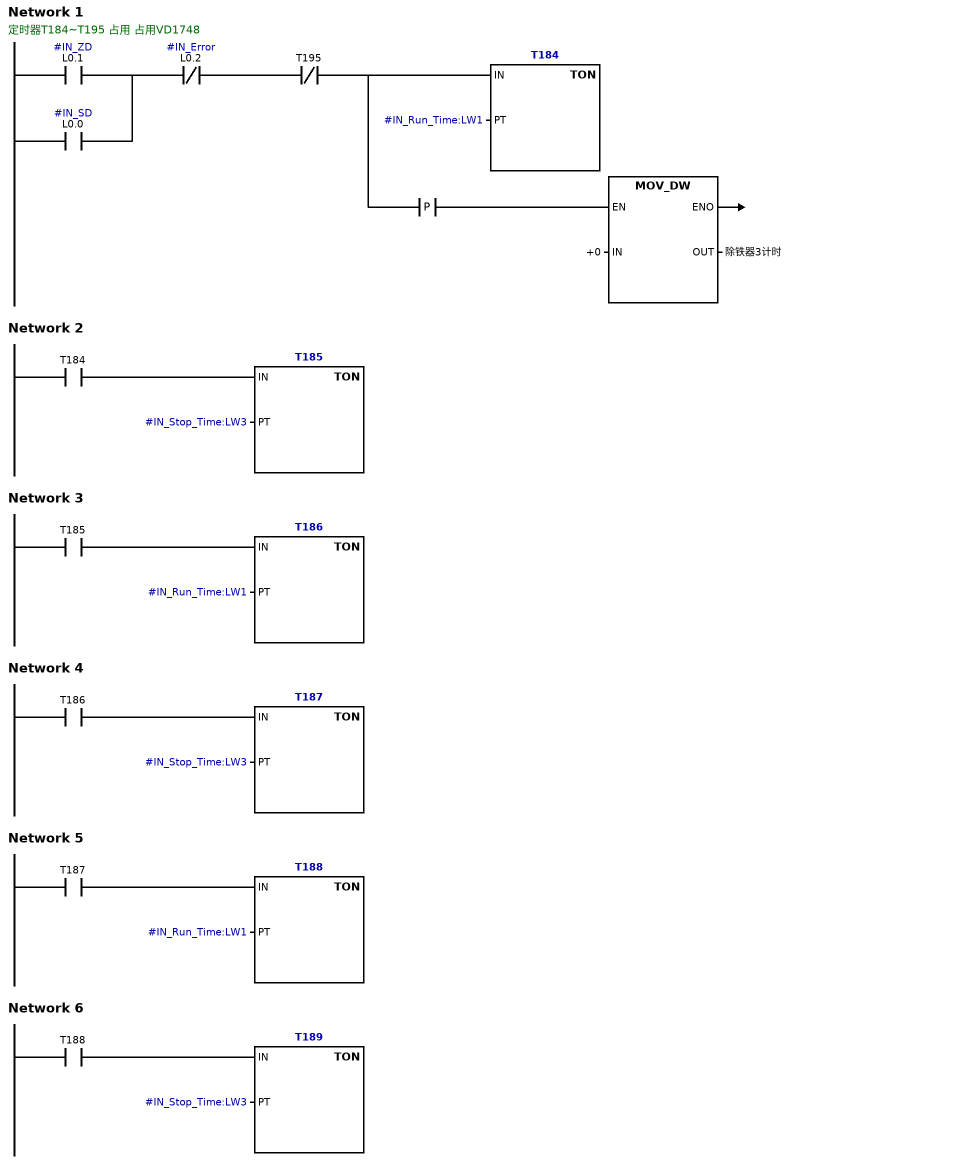
[picture p168: SBR79 networks 1-6]
Network 1
// 定时器T184~T195 占用 占用VD1748
// (network saved uncompiled; LAD cells follow)
// row 0: c0 -| |- #IN_ZD:L0.1 v  c1 -|/|- #IN_Error:L0.2  c2 -|/|- T195 v  c3 --  c4 [TON T184 IN:=power@row0, PT:=#IN_Run_Time:LW1]
// row 1: c0 -| |- #IN_SD:L0.0 ^  c2 ^v  c4 [box]
// row 2: c2 ^  c3 -|P|-  c4 --  c5 [MOV_DW EN:=power@row2, IN:=+0, ENO=>power, OUT=>除铁器3计时]  c6 ->
// row 3: c5 [box]
Network 2
LD     T184
TON    T185, #IN_Stop_Time:LW3
Network 3
LD     T185
TON    T186, #IN_Run_Time:LW1
Network 4
LD     T186
TON    T187, #IN_Stop_Time:LW3
Network 5
LD     T187
TON    T188, #IN_Run_Time:LW1
Network 6
LD     T188
TON    T189, #IN_Stop_Time:LW3
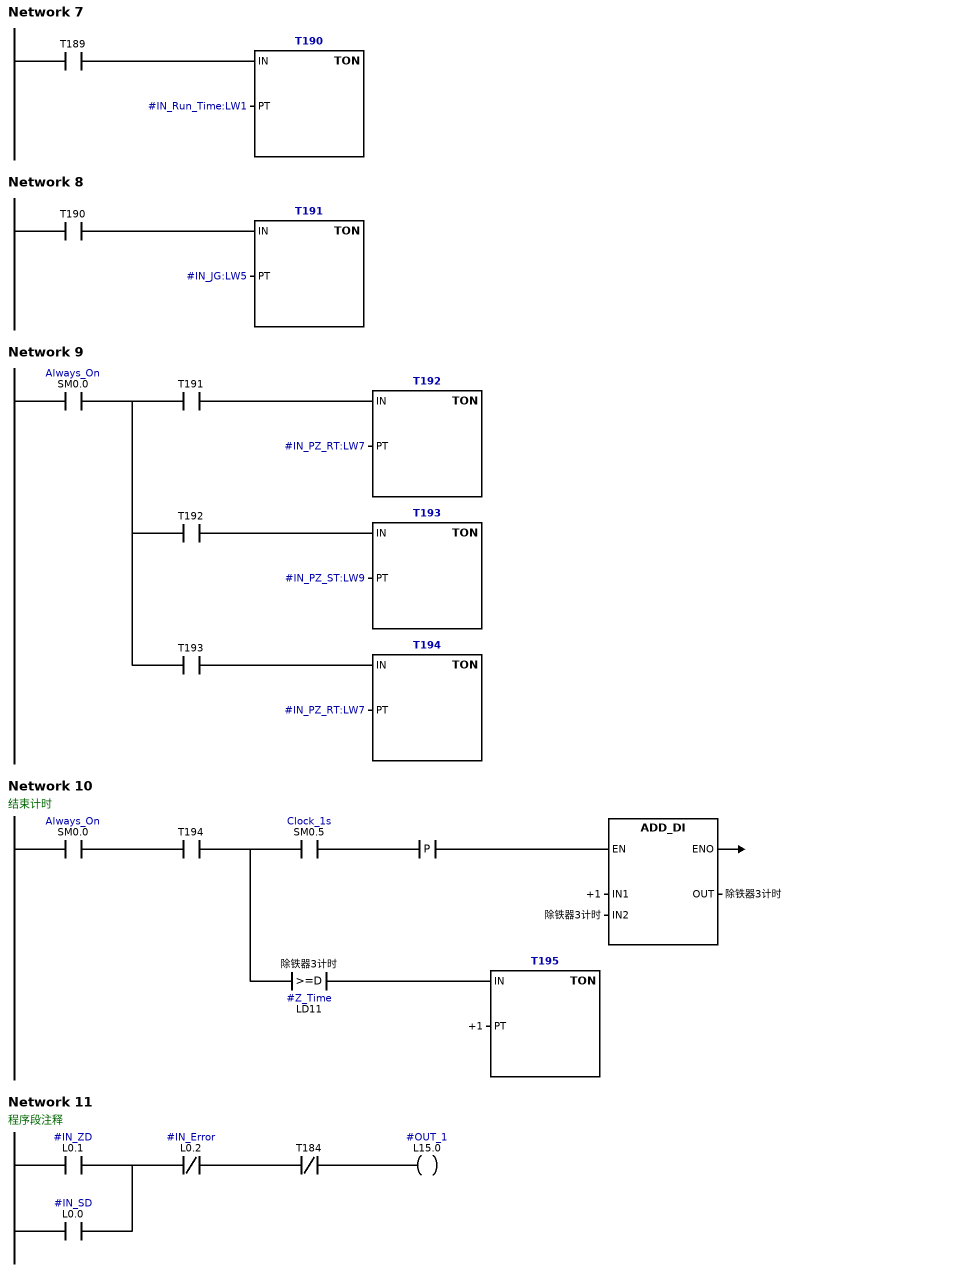
Network 7
LD     T189
TON    T190, #IN_Run_Time:LW1
Network 8
LD     T190
TON    T191, #IN_JG:LW5
Network 9
LD     Always_On:SM0.0
LPS
A      T191
TON    T192, #IN_PZ_RT:LW7
LRD
A      T192
TON    T193, #IN_PZ_ST:LW9
LPP
A      T193
TON    T194, #IN_PZ_RT:LW7
Network 10
// 结束计时
// (network saved uncompiled; LAD cells follow)
// row 0: c0 -| |- Always_On:SM0.0  c1 -| |- T194 v  c2 -| |- Clock_1s:SM0.5  c3 -|P|-  c4 --  c5 [ADD_DI EN:=power@row0, IN1:=+1, IN2:=除铁器3计时, ENO=>power, OUT=>除铁器3计时]  c6 ->
// row 1: c1 ^v  c5 [box]
// row 2: c1 ^  c2 -|>=D|- 除铁器3计时, #Z_Time:LD11  c3 --  c4 [TON T195 IN:=power@row2, PT:=+1]
// row 3: c4 [box]
Network 11
//  程序段注释
LD     #IN_ZD:L0.1
O      #IN_SD:L0.0
AN     #IN_Error:L0.2
AN     T184
=      #OUT_1:L15.0
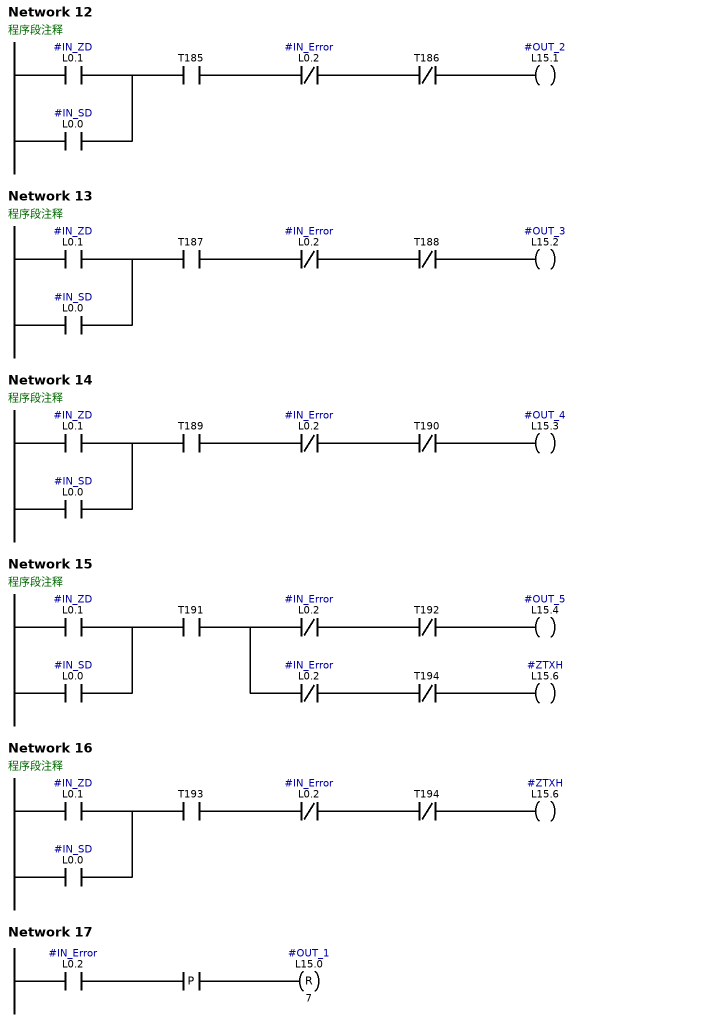
Network 12
//  程序段注释
LD     #IN_ZD:L0.1
O      #IN_SD:L0.0
A      T185
AN     #IN_Error:L0.2
AN     T186
=      #OUT_2:L15.1
Network 13
//  程序段注释
LD     #IN_ZD:L0.1
O      #IN_SD:L0.0
A      T187
AN     #IN_Error:L0.2
AN     T188
=      #OUT_3:L15.2
Network 14
//  程序段注释
LD     #IN_ZD:L0.1
O      #IN_SD:L0.0
A      T189
AN     #IN_Error:L0.2
AN     T190
=      #OUT_4:L15.3
Network 15
//  程序段注释
LD     #IN_ZD:L0.1
O      #IN_SD:L0.0
A      T191
LPS
AN     #IN_Error:L0.2
AN     T192
=      #OUT_5:L15.4
LPP
AN     #IN_Error:L0.2
AN     T194
=      #ZTXH:L15.6
Network 16
//  程序段注释
LD     #IN_ZD:L0.1
O      #IN_SD:L0.0
A      T193
AN     #IN_Error:L0.2
AN     T194
=      #ZTXH:L15.6
Network 17
LD     #IN_Error:L0.2
EU
R      #OUT_1:L15.0, 7
END_SUBROUTINE_BLOCK

SUBROUTINE_BLOCK 脉冲阀4组1:SBR80
TITLE=
VAR_INPUT
IN_SD:BOOL;	// L0.0 
IN_ZD:BOOL;	// L0.1 
IN_Error:BOOL;	// L0.2 
IN_Run_Time:INT;	// LW1 
IN_Stop_Time:INT;	// LW3 
END_VAR
VAR_OUTPUT
OUT_1:BOOL;	// L5.0 
OUT_2:BOOL;	// L5.1 
OUT_3:BOOL;	// L5.2 
OUT_4:BOOL;	// L5.3 
END_VAR
VAR
TP1:BOOL;	// L5.4 
TP2:BOOL;	// L5.5 
END_VAR
BEGIN
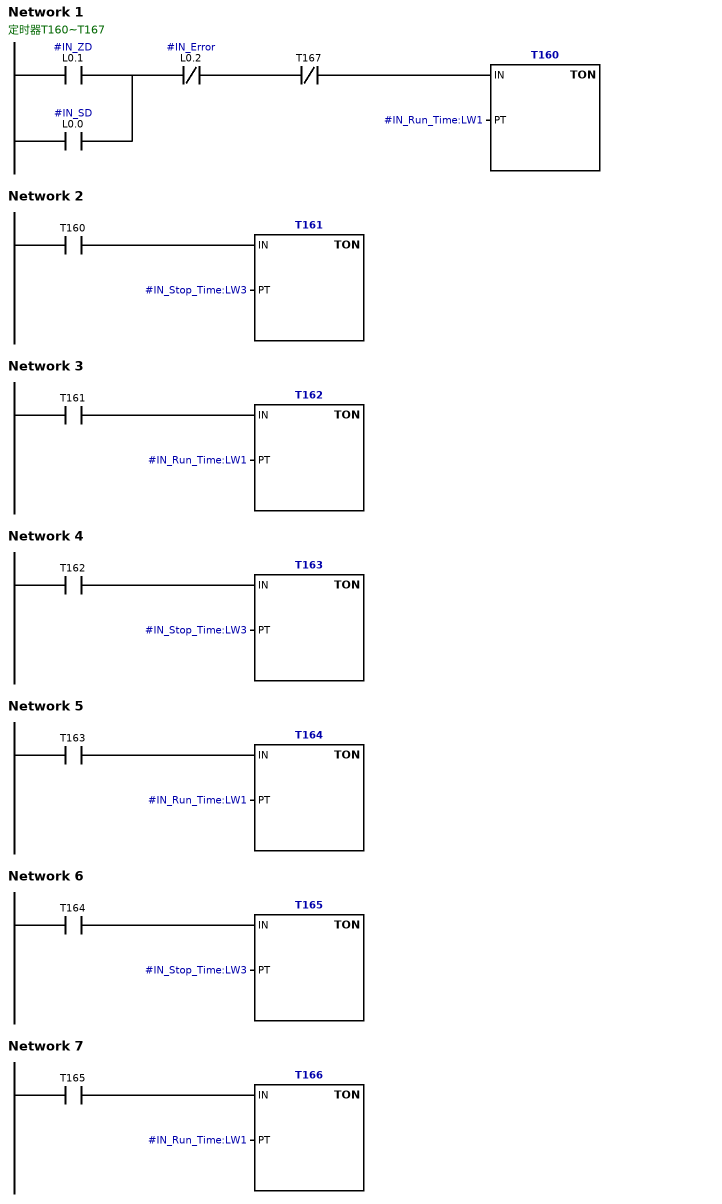
Network 1
// 定时器T160~T167
LD     #IN_ZD:L0.1
O      #IN_SD:L0.0
AN     #IN_Error:L0.2
AN     T167
TON    T160, #IN_Run_Time:LW1
Network 2
LD     T160
TON    T161, #IN_Stop_Time:LW3
Network 3
LD     T161
TON    T162, #IN_Run_Time:LW1
Network 4
LD     T162
TON    T163, #IN_Stop_Time:LW3
Network 5
LD     T163
TON    T164, #IN_Run_Time:LW1
Network 6
LD     T164
TON    T165, #IN_Stop_Time:LW3
Network 7
LD     T165
TON    T166, #IN_Run_Time:LW1
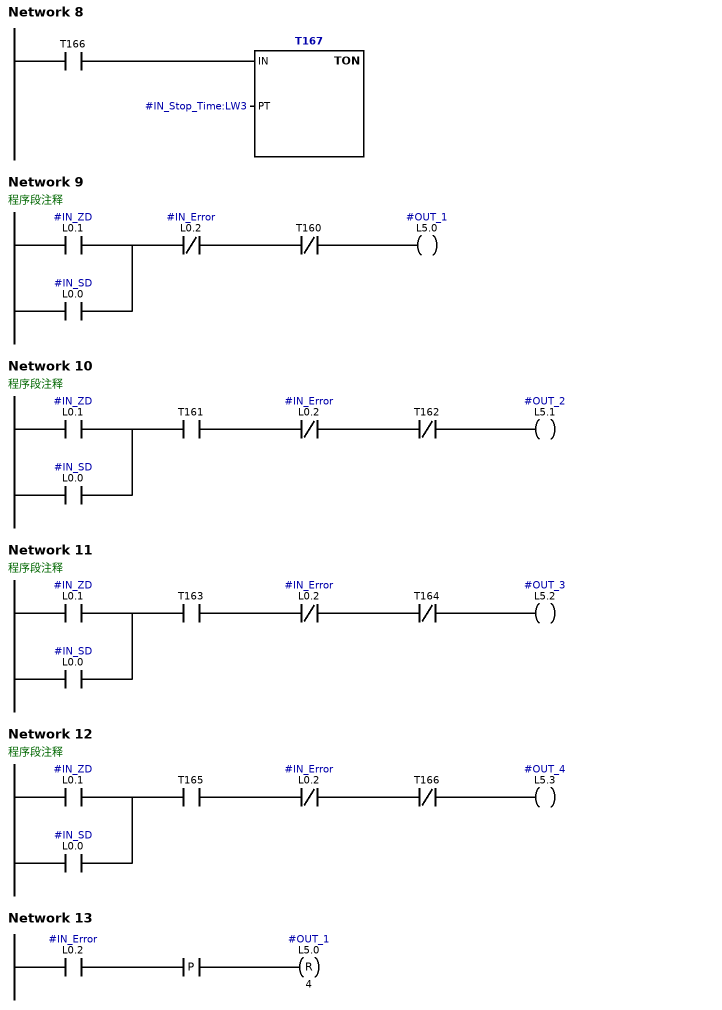
Network 8
LD     T166
TON    T167, #IN_Stop_Time:LW3
Network 9
//  程序段注释
LD     #IN_ZD:L0.1
O      #IN_SD:L0.0
AN     #IN_Error:L0.2
AN     T160
=      #OUT_1:L5.0
Network 10
//  程序段注释
LD     #IN_ZD:L0.1
O      #IN_SD:L0.0
A      T161
AN     #IN_Error:L0.2
AN     T162
=      #OUT_2:L5.1
Network 11
//  程序段注释
LD     #IN_ZD:L0.1
O      #IN_SD:L0.0
A      T163
AN     #IN_Error:L0.2
AN     T164
=      #OUT_3:L5.2
Network 12
//  程序段注释
LD     #IN_ZD:L0.1
O      #IN_SD:L0.0
A      T165
AN     #IN_Error:L0.2
AN     T166
=      #OUT_4:L5.3
Network 13
LD     #IN_Error:L0.2
EU
R      #OUT_1:L5.0, 4
END_SUBROUTINE_BLOCK

SUBROUTINE_BLOCK 脉冲阀4组2:SBR81
TITLE=
VAR_INPUT
IN_SD:BOOL;	// L0.0 
IN_ZD:BOOL;	// L0.1 
IN_Error:BOOL;	// L0.2 
IN_Run_Time:INT;	// LW1 
IN_Stop_Time:INT;	// LW3 
END_VAR
VAR_OUTPUT
OUT_1:BOOL;	// L5.0 
OUT_2:BOOL;	// L5.1 
OUT_3:BOOL;	// L5.2 
OUT_4:BOOL;	// L5.3 
END_VAR
VAR
TP1:BOOL;	// L5.4 
TP2:BOOL;	// L5.5 
END_VAR
BEGIN
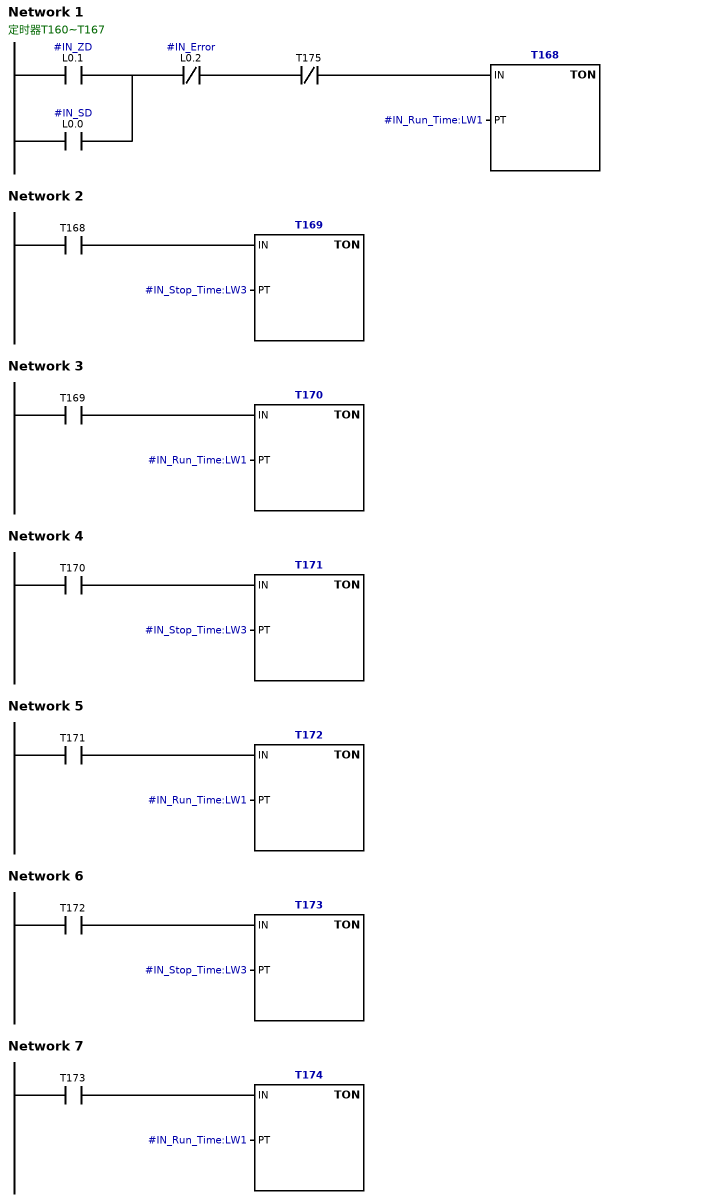
Network 1
// 定时器T160~T167
LD     #IN_ZD:L0.1
O      #IN_SD:L0.0
AN     #IN_Error:L0.2
AN     T175
TON    T168, #IN_Run_Time:LW1
Network 2
LD     T168
TON    T169, #IN_Stop_Time:LW3
Network 3
LD     T169
TON    T170, #IN_Run_Time:LW1
Network 4
LD     T170
TON    T171, #IN_Stop_Time:LW3
Network 5
LD     T171
TON    T172, #IN_Run_Time:LW1
Network 6
LD     T172
TON    T173, #IN_Stop_Time:LW3
Network 7
LD     T173
TON    T174, #IN_Run_Time:LW1
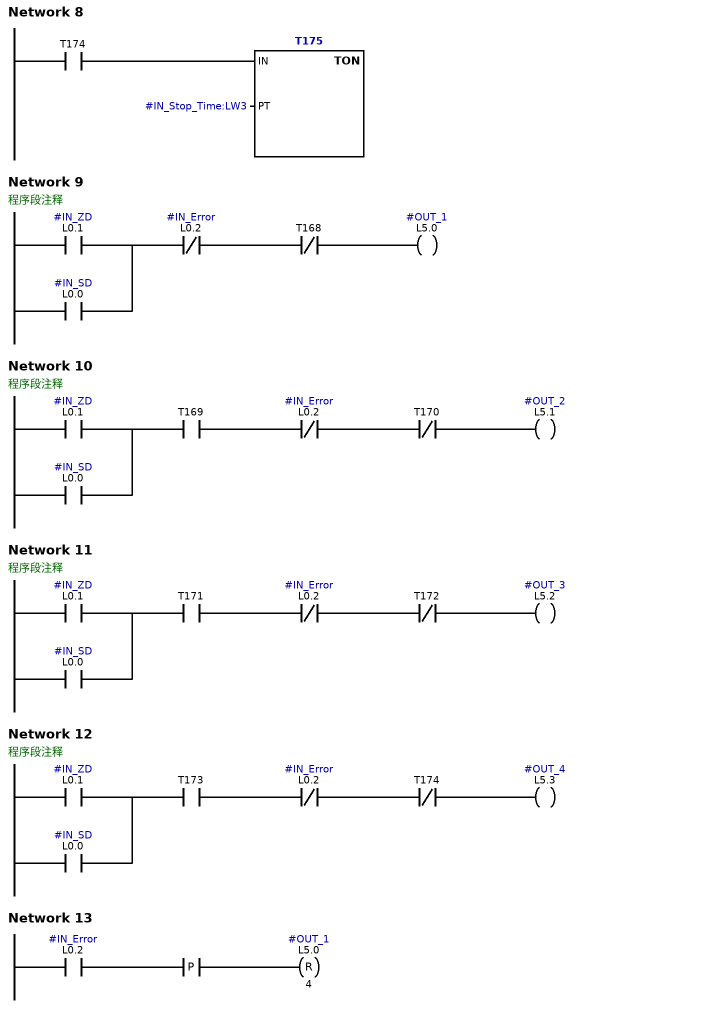
Network 8
LD     T174
TON    T175, #IN_Stop_Time:LW3
Network 9
//  程序段注释
LD     #IN_ZD:L0.1
O      #IN_SD:L0.0
AN     #IN_Error:L0.2
AN     T168
=      #OUT_1:L5.0
Network 10
//  程序段注释
LD     #IN_ZD:L0.1
O      #IN_SD:L0.0
A      T169
AN     #IN_Error:L0.2
AN     T170
=      #OUT_2:L5.1
Network 11
//  程序段注释
LD     #IN_ZD:L0.1
O      #IN_SD:L0.0
A      T171
AN     #IN_Error:L0.2
AN     T172
=      #OUT_3:L5.2
Network 12
//  程序段注释
LD     #IN_ZD:L0.1
O      #IN_SD:L0.0
A      T173
AN     #IN_Error:L0.2
AN     T174
=      #OUT_4:L5.3
Network 13
LD     #IN_Error:L0.2
EU
R      #OUT_1:L5.0, 4
END_SUBROUTINE_BLOCK

SUBROUTINE_BLOCK 脉冲阀4组3:SBR82
TITLE=
VAR_INPUT
IN_SD:BOOL;	// L0.0 
IN_ZD:BOOL;	// L0.1 
IN_Error:BOOL;	// L0.2 
IN_Run_Time:INT;	// LW1 
IN_Stop_Time:INT;	// LW3 
END_VAR
VAR_OUTPUT
OUT_1:BOOL;	// L5.0 
OUT_2:BOOL;	// L5.1 
OUT_3:BOOL;	// L5.2 
OUT_4:BOOL;	// L5.3 
END_VAR
VAR
TP1:BOOL;	// L5.4 
TP2:BOOL;	// L5.5 
END_VAR
BEGIN
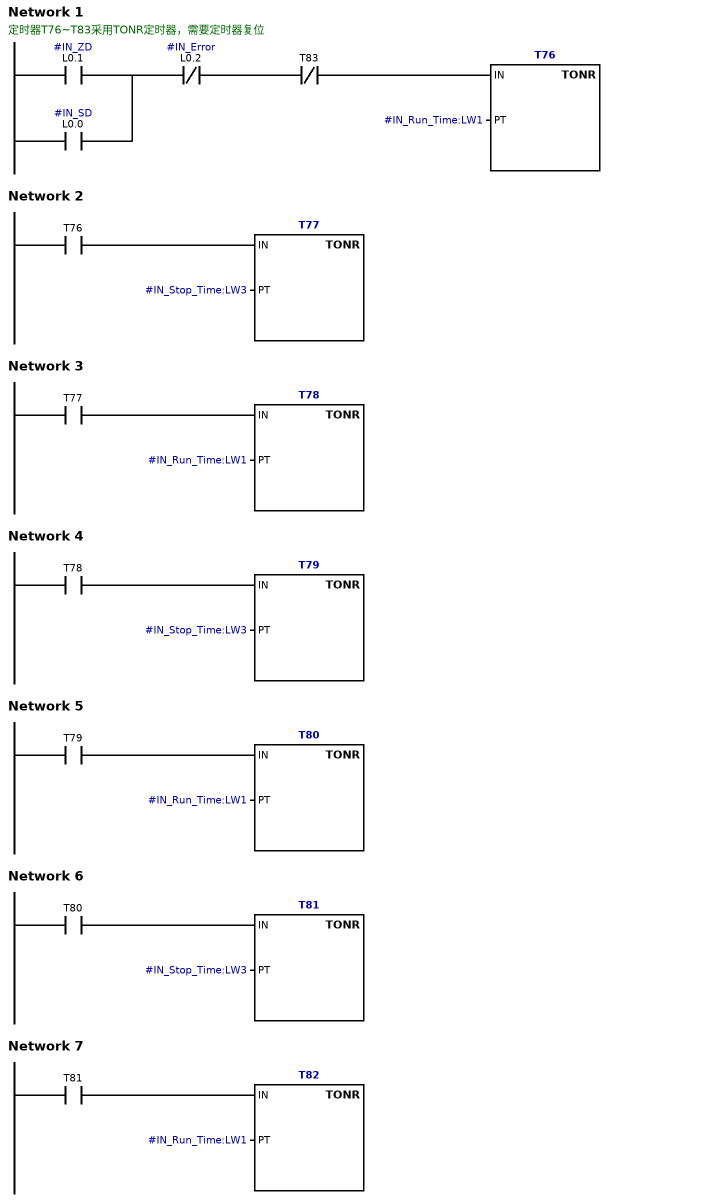
Network 1
// 定时器T76~T83采用TONR定时器，需要定时器复位
LD     #IN_ZD:L0.1
O      #IN_SD:L0.0
AN     #IN_Error:L0.2
AN     T83
TONR   T76, #IN_Run_Time:LW1
Network 2
LD     T76
TONR   T77, #IN_Stop_Time:LW3
Network 3
LD     T77
TONR   T78, #IN_Run_Time:LW1
Network 4
LD     T78
TONR   T79, #IN_Stop_Time:LW3
Network 5
LD     T79
TONR   T80, #IN_Run_Time:LW1
Network 6
LD     T80
TONR   T81, #IN_Stop_Time:LW3
Network 7
LD     T81
TONR   T82, #IN_Run_Time:LW1
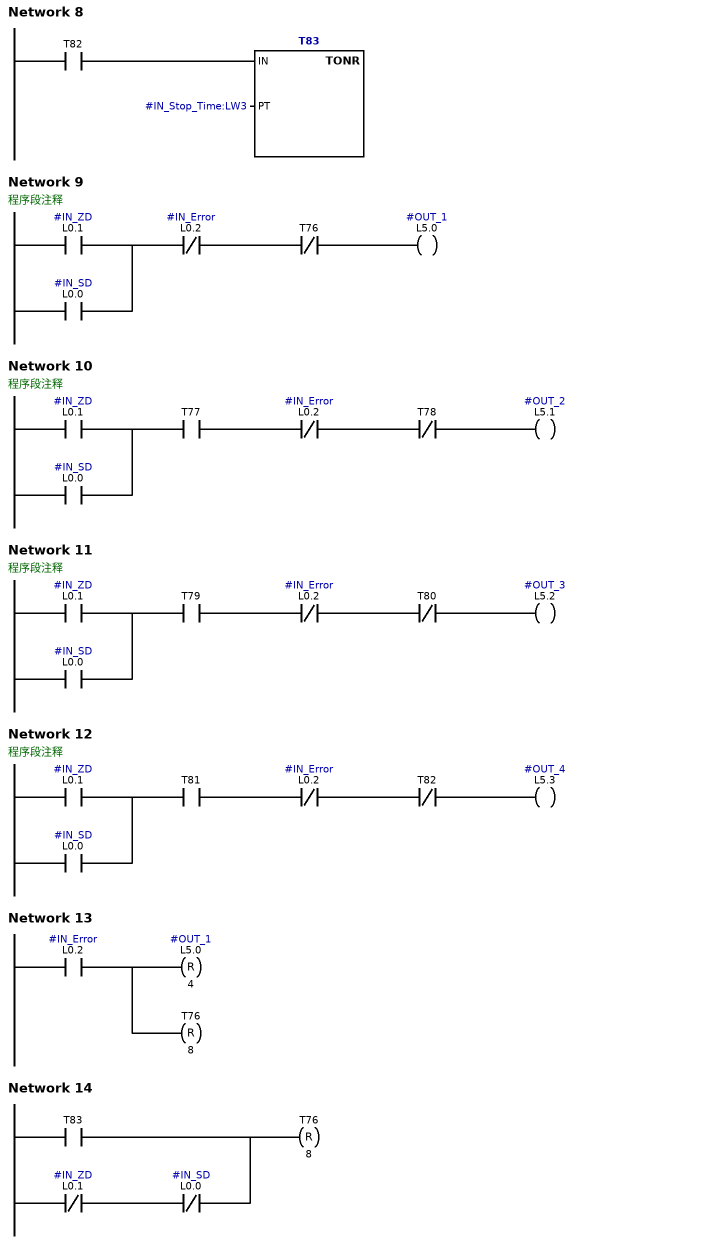
Network 8
LD     T82
TONR   T83, #IN_Stop_Time:LW3
Network 9
//  程序段注释
LD     #IN_ZD:L0.1
O      #IN_SD:L0.0
AN     #IN_Error:L0.2
AN     T76
=      #OUT_1:L5.0
Network 10
//  程序段注释
LD     #IN_ZD:L0.1
O      #IN_SD:L0.0
A      T77
AN     #IN_Error:L0.2
AN     T78
=      #OUT_2:L5.1
Network 11
//  程序段注释
LD     #IN_ZD:L0.1
O      #IN_SD:L0.0
A      T79
AN     #IN_Error:L0.2
AN     T80
=      #OUT_3:L5.2
Network 12
//  程序段注释
LD     #IN_ZD:L0.1
O      #IN_SD:L0.0
A      T81
AN     #IN_Error:L0.2
AN     T82
=      #OUT_4:L5.3
Network 13
LD     #IN_Error:L0.2
R      #OUT_1:L5.0, 4
R      T76, 8
Network 14
LD     T83
LDN    #IN_ZD:L0.1
AN     #IN_SD:L0.0
OLD
R      T76, 8
END_SUBROUTINE_BLOCK

SUBROUTINE_BLOCK 脉冲阀4组4:SBR83
TITLE=
VAR_INPUT
IN_SD:BOOL;	// L0.0 
IN_ZD:BOOL;	// L0.1 
IN_Error:BOOL;	// L0.2 
IN_Run_Time:INT;	// LW1 
IN_Stop_Time:INT;	// LW3 
END_VAR
VAR_OUTPUT
OUT_1:BOOL;	// L5.0 
OUT_2:BOOL;	// L5.1 
OUT_3:BOOL;	// L5.2 
OUT_4:BOOL;	// L5.3 
END_VAR
VAR
TP1:BOOL;	// L5.4 
TP2:BOOL;	// L5.5 
END_VAR
BEGIN
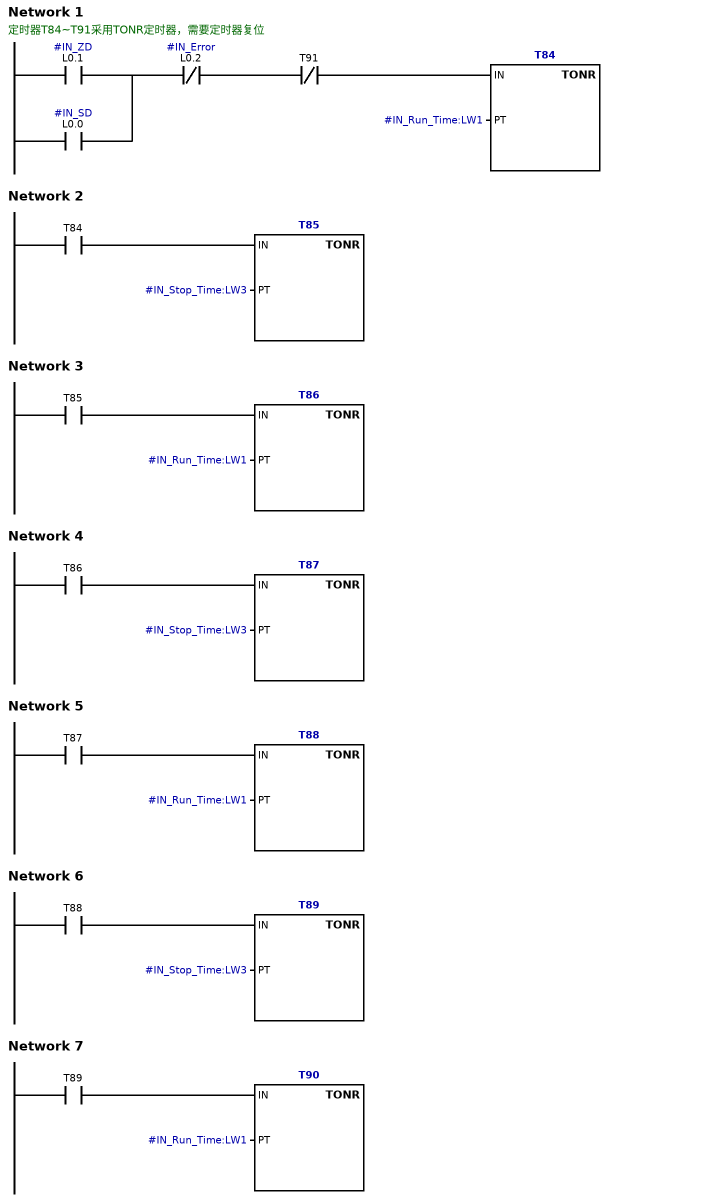
Network 1
// 定时器T84~T91采用TONR定时器，需要定时器复位
LD     #IN_ZD:L0.1
O      #IN_SD:L0.0
AN     #IN_Error:L0.2
AN     T91
TONR   T84, #IN_Run_Time:LW1
Network 2
LD     T84
TONR   T85, #IN_Stop_Time:LW3
Network 3
LD     T85
TONR   T86, #IN_Run_Time:LW1
Network 4
LD     T86
TONR   T87, #IN_Stop_Time:LW3
Network 5
LD     T87
TONR   T88, #IN_Run_Time:LW1
Network 6
LD     T88
TONR   T89, #IN_Stop_Time:LW3
Network 7
LD     T89
TONR   T90, #IN_Run_Time:LW1
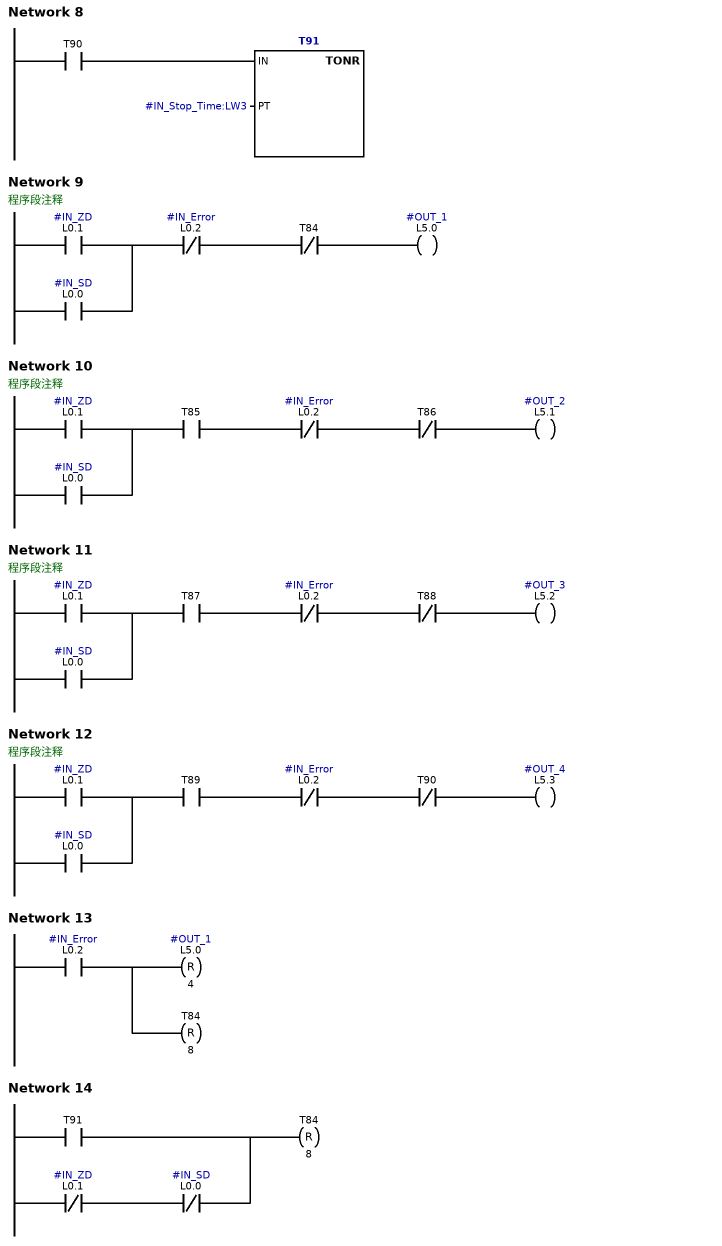
Network 8
LD     T90
TONR   T91, #IN_Stop_Time:LW3
Network 9
//  程序段注释
LD     #IN_ZD:L0.1
O      #IN_SD:L0.0
AN     #IN_Error:L0.2
AN     T84
=      #OUT_1:L5.0
Network 10
//  程序段注释
LD     #IN_ZD:L0.1
O      #IN_SD:L0.0
A      T85
AN     #IN_Error:L0.2
AN     T86
=      #OUT_2:L5.1
Network 11
//  程序段注释
LD     #IN_ZD:L0.1
O      #IN_SD:L0.0
A      T87
AN     #IN_Error:L0.2
AN     T88
=      #OUT_3:L5.2
Network 12
//  程序段注释
LD     #IN_ZD:L0.1
O      #IN_SD:L0.0
A      T89
AN     #IN_Error:L0.2
AN     T90
=      #OUT_4:L5.3
Network 13
LD     #IN_Error:L0.2
R      #OUT_1:L5.0, 4
R      T84, 8
Network 14
LD     T91
LDN    #IN_ZD:L0.1
AN     #IN_SD:L0.0
OLD
R      T84, 8
END_SUBROUTINE_BLOCK

SUBROUTINE_BLOCK 脉冲阀4组5:SBR84
TITLE=
VAR_INPUT
IN_SD:BOOL;	// L0.0 
IN_ZD:BOOL;	// L0.1 
IN_Error:BOOL;	// L0.2 
IN_Run_Time:INT;	// LW1 
IN_Stop_Time:INT;	// LW3 
END_VAR
VAR_OUTPUT
OUT_1:BOOL;	// L5.0 
OUT_2:BOOL;	// L5.1 
OUT_3:BOOL;	// L5.2 
OUT_4:BOOL;	// L5.3 
END_VAR
VAR
TP1:BOOL;	// L5.4 
TP2:BOOL;	// L5.5 
END_VAR
BEGIN
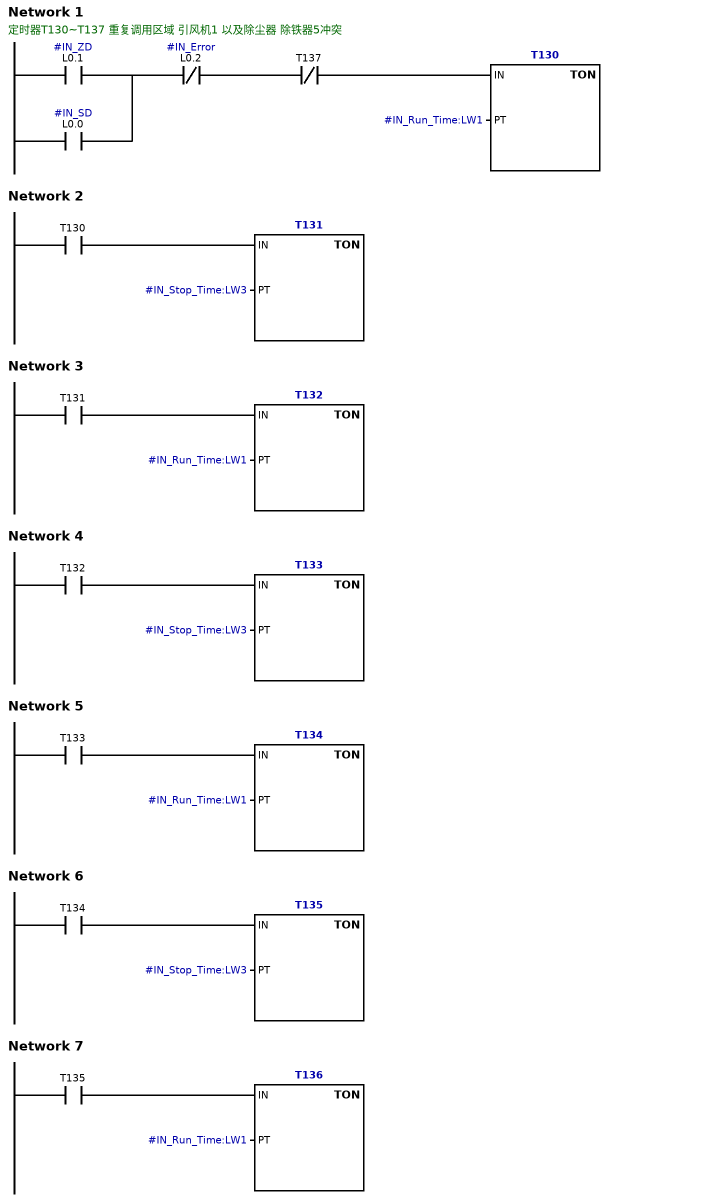
Network 1
// 定时器T130~T137 重复调用区域 引风机1 以及除尘器 除铁器5冲突
LD     #IN_ZD:L0.1
O      #IN_SD:L0.0
AN     #IN_Error:L0.2
AN     T137
TON    T130, #IN_Run_Time:LW1
Network 2
LD     T130
TON    T131, #IN_Stop_Time:LW3
Network 3
LD     T131
TON    T132, #IN_Run_Time:LW1
Network 4
LD     T132
TON    T133, #IN_Stop_Time:LW3
Network 5
LD     T133
TON    T134, #IN_Run_Time:LW1
Network 6
LD     T134
TON    T135, #IN_Stop_Time:LW3
Network 7
LD     T135
TON    T136, #IN_Run_Time:LW1
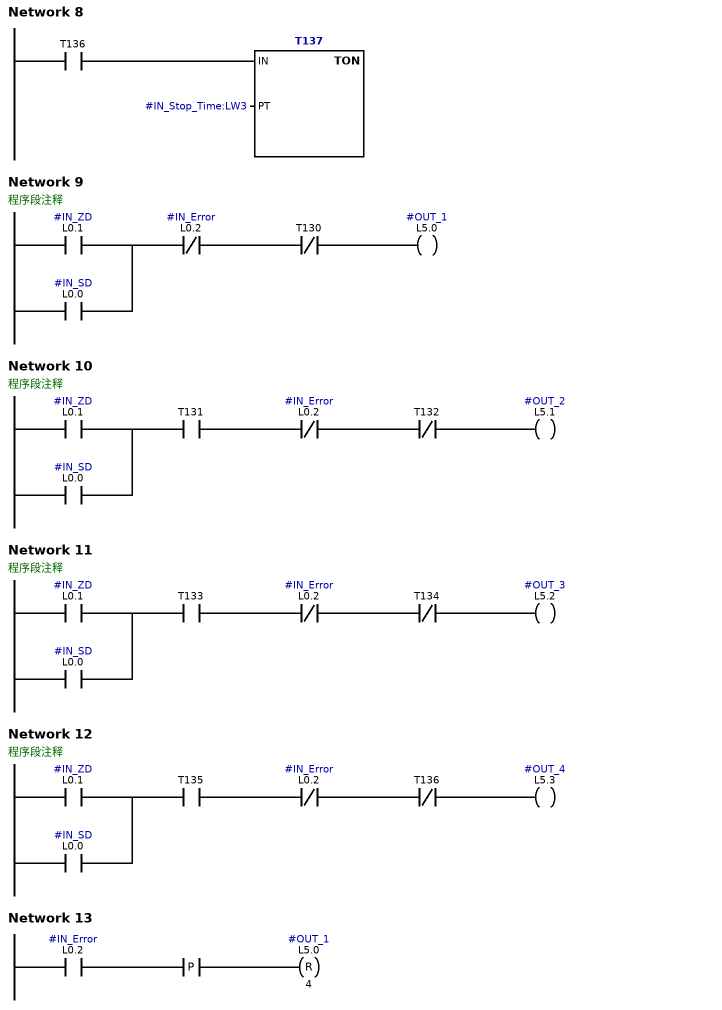
Network 8
LD     T136
TON    T137, #IN_Stop_Time:LW3
Network 9
//  程序段注释
LD     #IN_ZD:L0.1
O      #IN_SD:L0.0
AN     #IN_Error:L0.2
AN     T130
=      #OUT_1:L5.0
Network 10
//  程序段注释
LD     #IN_ZD:L0.1
O      #IN_SD:L0.0
A      T131
AN     #IN_Error:L0.2
AN     T132
=      #OUT_2:L5.1
Network 11
//  程序段注释
LD     #IN_ZD:L0.1
O      #IN_SD:L0.0
A      T133
AN     #IN_Error:L0.2
AN     T134
=      #OUT_3:L5.2
Network 12
//  程序段注释
LD     #IN_ZD:L0.1
O      #IN_SD:L0.0
A      T135
AN     #IN_Error:L0.2
AN     T136
=      #OUT_4:L5.3
Network 13
LD     #IN_Error:L0.2
EU
R      #OUT_1:L5.0, 4
END_SUBROUTINE_BLOCK

SUBROUTINE_BLOCK 除铁器4组1:SBR85
TITLE=
VAR_INPUT
IN_SD:BOOL;	// L0.0 
IN_ZD:BOOL;	// L0.1 
IN_Error:BOOL;	// L0.2 
IN_Run_Time:INT;	// LW1 
IN_Stop_Time:INT;	// LW3 
Z_Time:DINT;	// LD5 
END_VAR
VAR_IN_OUT
JS:DINT;	// LD9 
END_VAR
VAR_OUTPUT
OUT_1:BOOL;	// L13.0 
OUT_2:BOOL;	// L13.1 
OUT_3:BOOL;	// L13.2 
OUT_4:BOOL;	// L13.3 
END_VAR
VAR
TP1:BOOL;	// L13.4 
TP2:BOOL;	// L13.5 
END_VAR
BEGIN
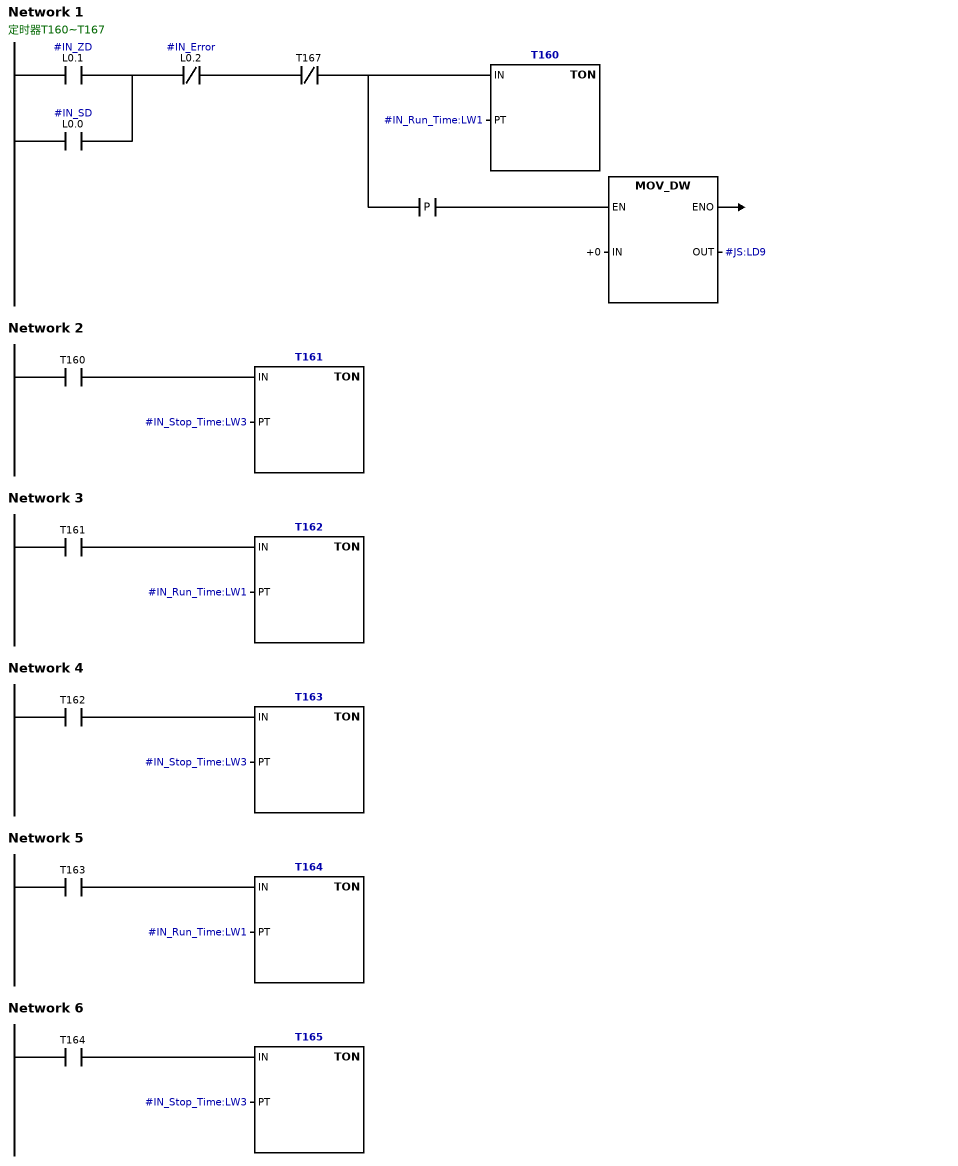
Network 1
// 定时器T160~T167
LD     #IN_ZD:L0.1
O      #IN_SD:L0.0
AN     #IN_Error:L0.2
AN     T167
TON    T160, #IN_Run_Time:LW1
EU
MOVD   +0, #JS:LD9
Network 2
LD     T160
TON    T161, #IN_Stop_Time:LW3
Network 3
LD     T161
TON    T162, #IN_Run_Time:LW1
Network 4
LD     T162
TON    T163, #IN_Stop_Time:LW3
Network 5
LD     T163
TON    T164, #IN_Run_Time:LW1
Network 6
LD     T164
TON    T165, #IN_Stop_Time:LW3
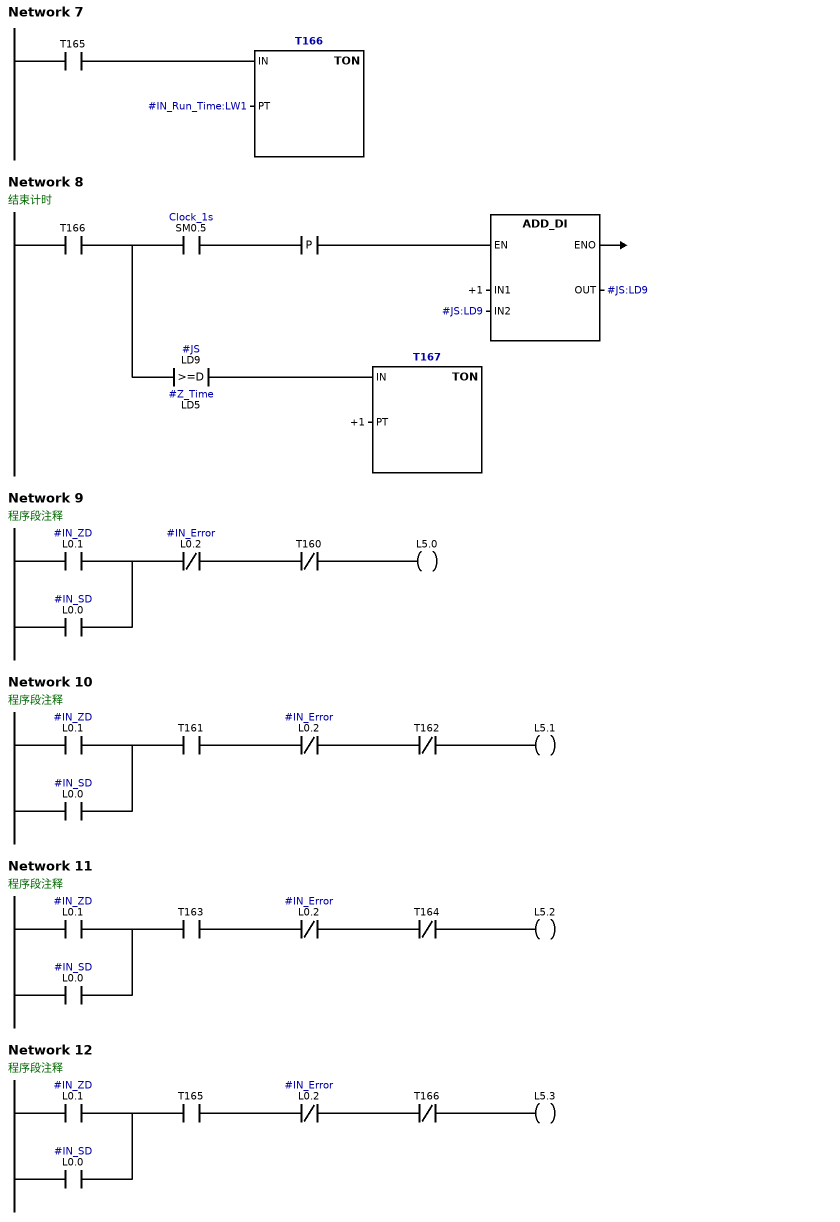
Network 7
LD     T165
TON    T166, #IN_Run_Time:LW1
Network 8
// 结束计时
LD     T166
LPS
A      Clock_1s:SM0.5
EU
+D     +1, #JS:LD9
LPP
AD>=   #JS:LD9, #Z_Time:LD5
TON    T167, +1
Network 9
//  程序段注释
LD     #IN_ZD:L0.1
O      #IN_SD:L0.0
AN     #IN_Error:L0.2
AN     T160
=      L5.0
Network 10
//  程序段注释
LD     #IN_ZD:L0.1
O      #IN_SD:L0.0
A      T161
AN     #IN_Error:L0.2
AN     T162
=      L5.1
Network 11
//  程序段注释
LD     #IN_ZD:L0.1
O      #IN_SD:L0.0
A      T163
AN     #IN_Error:L0.2
AN     T164
=      L5.2
Network 12
//  程序段注释
LD     #IN_ZD:L0.1
O      #IN_SD:L0.0
A      T165
AN     #IN_Error:L0.2
AN     T166
=      L5.3
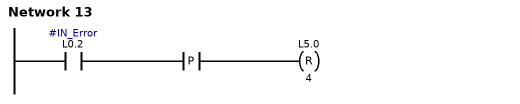
Network 13
LD     #IN_Error:L0.2
EU
R      L5.0, 4
END_SUBROUTINE_BLOCK

SUBROUTINE_BLOCK 除铁器4组2:SBR86
TITLE=
VAR_INPUT
IN_SD:BOOL;	// L0.0 
IN_ZD:BOOL;	// L0.1 
IN_Error:BOOL;	// L0.2 
IN_Run_Time:INT;	// LW1 
IN_Stop_Time:INT;	// LW3 
Z_Time:DINT;	// LD5 
END_VAR
VAR_IN_OUT
JS:DINT;	// LD9 
END_VAR
VAR_OUTPUT
OUT_1:BOOL;	// L13.0 
OUT_2:BOOL;	// L13.1 
OUT_3:BOOL;	// L13.2 
OUT_4:BOOL;	// L13.3 
END_VAR
VAR
TP1:BOOL;	// L13.4 
TP2:BOOL;	// L13.5 
END_VAR
BEGIN
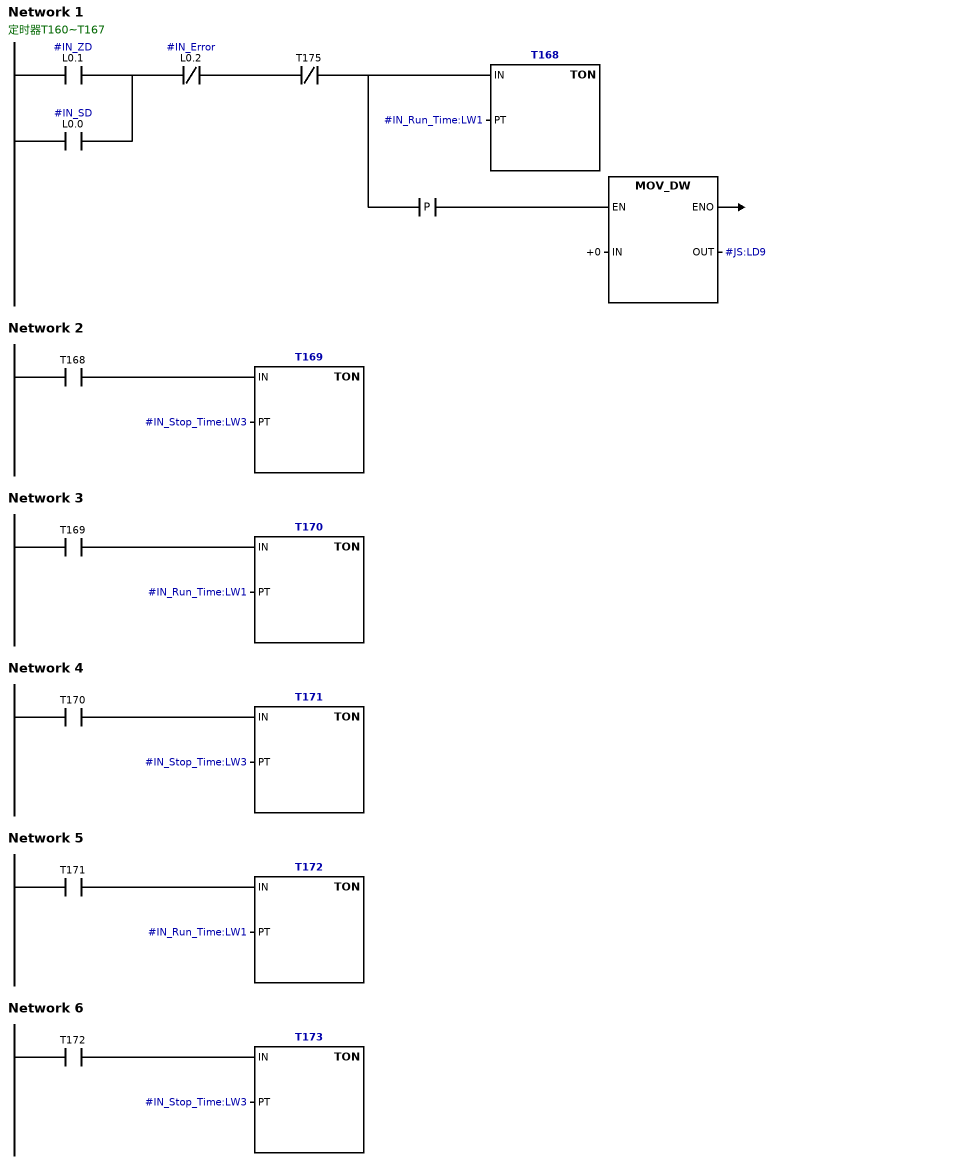
Network 1
// 定时器T160~T167
LD     #IN_ZD:L0.1
O      #IN_SD:L0.0
AN     #IN_Error:L0.2
AN     T175
TON    T168, #IN_Run_Time:LW1
EU
MOVD   +0, #JS:LD9
Network 2
LD     T168
TON    T169, #IN_Stop_Time:LW3
Network 3
LD     T169
TON    T170, #IN_Run_Time:LW1
Network 4
LD     T170
TON    T171, #IN_Stop_Time:LW3
Network 5
LD     T171
TON    T172, #IN_Run_Time:LW1
Network 6
LD     T172
TON    T173, #IN_Stop_Time:LW3
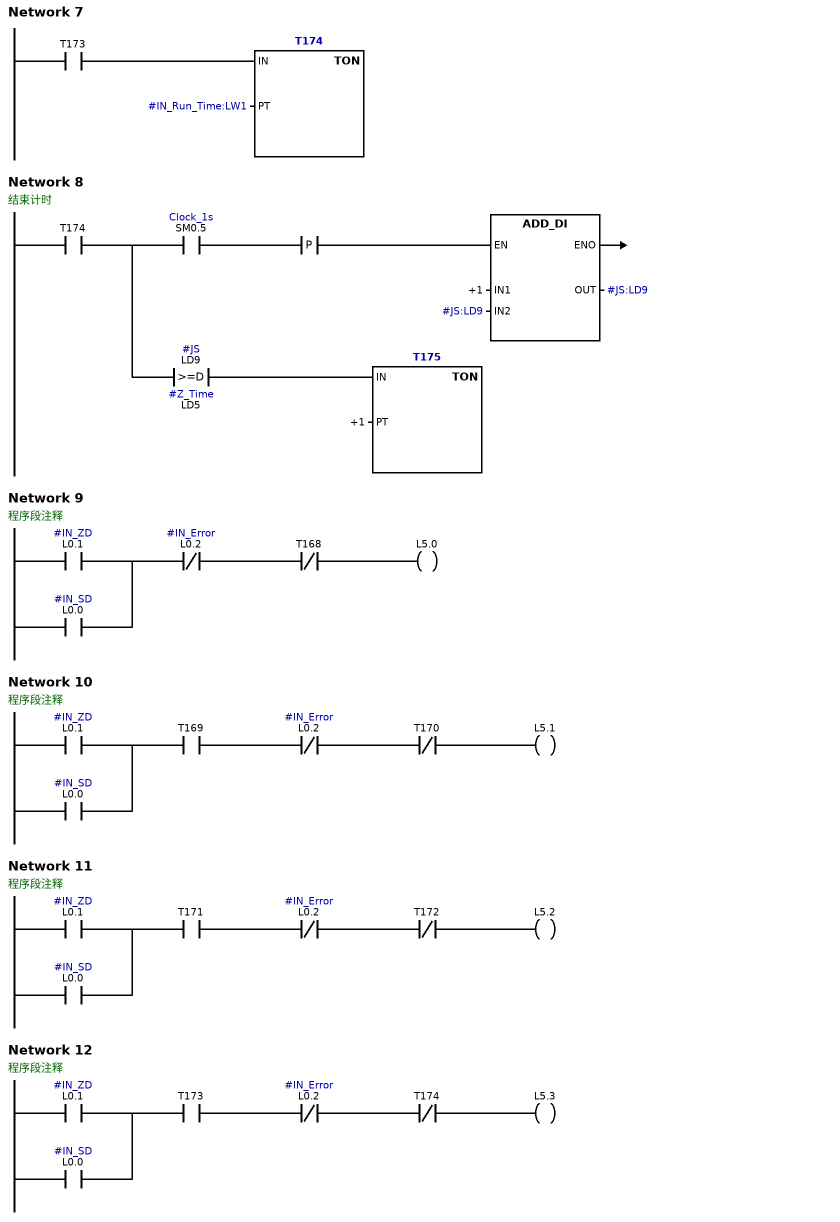
Network 7
LD     T173
TON    T174, #IN_Run_Time:LW1
Network 8
// 结束计时
LD     T174
LPS
A      Clock_1s:SM0.5
EU
+D     +1, #JS:LD9
LPP
AD>=   #JS:LD9, #Z_Time:LD5
TON    T175, +1
Network 9
//  程序段注释
LD     #IN_ZD:L0.1
O      #IN_SD:L0.0
AN     #IN_Error:L0.2
AN     T168
=      L5.0
Network 10
//  程序段注释
LD     #IN_ZD:L0.1
O      #IN_SD:L0.0
A      T169
AN     #IN_Error:L0.2
AN     T170
=      L5.1
Network 11
//  程序段注释
LD     #IN_ZD:L0.1
O      #IN_SD:L0.0
A      T171
AN     #IN_Error:L0.2
AN     T172
=      L5.2
Network 12
//  程序段注释
LD     #IN_ZD:L0.1
O      #IN_SD:L0.0
A      T173
AN     #IN_Error:L0.2
AN     T174
=      L5.3
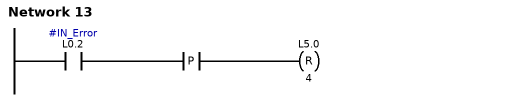
Network 13
LD     #IN_Error:L0.2
EU
R      L5.0, 4
END_SUBROUTINE_BLOCK

SUBROUTINE_BLOCK 除铁器4组3:SBR87
TITLE=
VAR_INPUT
IN_SD:BOOL;	// L0.0 
IN_ZD:BOOL;	// L0.1 
IN_Error:BOOL;	// L0.2 
IN_Run_Time:INT;	// LW1 
IN_Stop_Time:INT;	// LW3 
Z_Time:DINT;	// LD5 
END_VAR
VAR_IN_OUT
JS:DINT;	// LD9 
END_VAR
VAR_OUTPUT
OUT_1:BOOL;	// L13.0 
OUT_2:BOOL;	// L13.1 
OUT_3:BOOL;	// L13.2 
OUT_4:BOOL;	// L13.3 
END_VAR
VAR
TP1:BOOL;	// L13.4 
TP2:BOOL;	// L13.5 
END_VAR
BEGIN
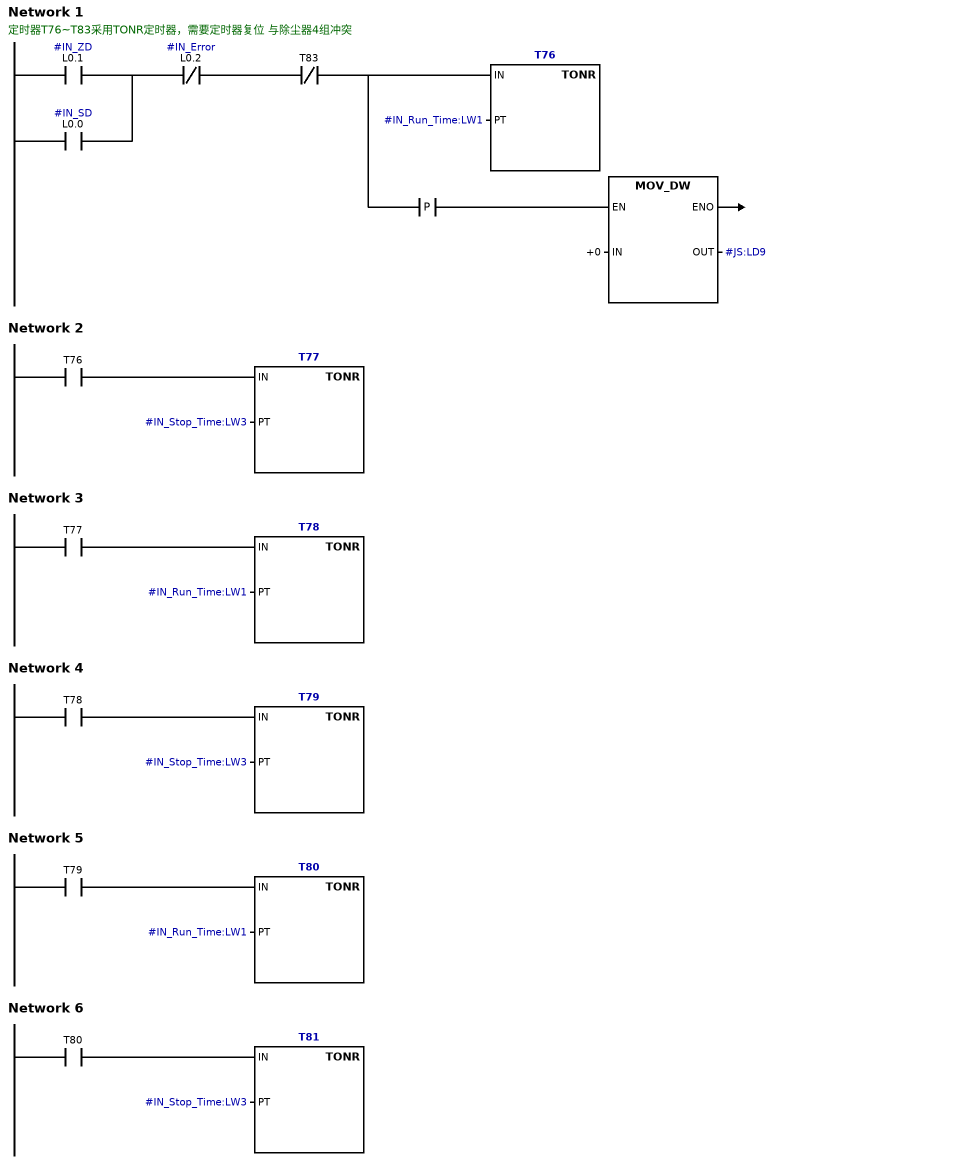
Network 1
// 定时器T76~T83采用TONR定时器，需要定时器复位 与除尘器4组冲突
LD     #IN_ZD:L0.1
O      #IN_SD:L0.0
AN     #IN_Error:L0.2
AN     T83
TONR   T76, #IN_Run_Time:LW1
EU
MOVD   +0, #JS:LD9
Network 2
LD     T76
TONR   T77, #IN_Stop_Time:LW3
Network 3
LD     T77
TONR   T78, #IN_Run_Time:LW1
Network 4
LD     T78
TONR   T79, #IN_Stop_Time:LW3
Network 5
LD     T79
TONR   T80, #IN_Run_Time:LW1
Network 6
LD     T80
TONR   T81, #IN_Stop_Time:LW3
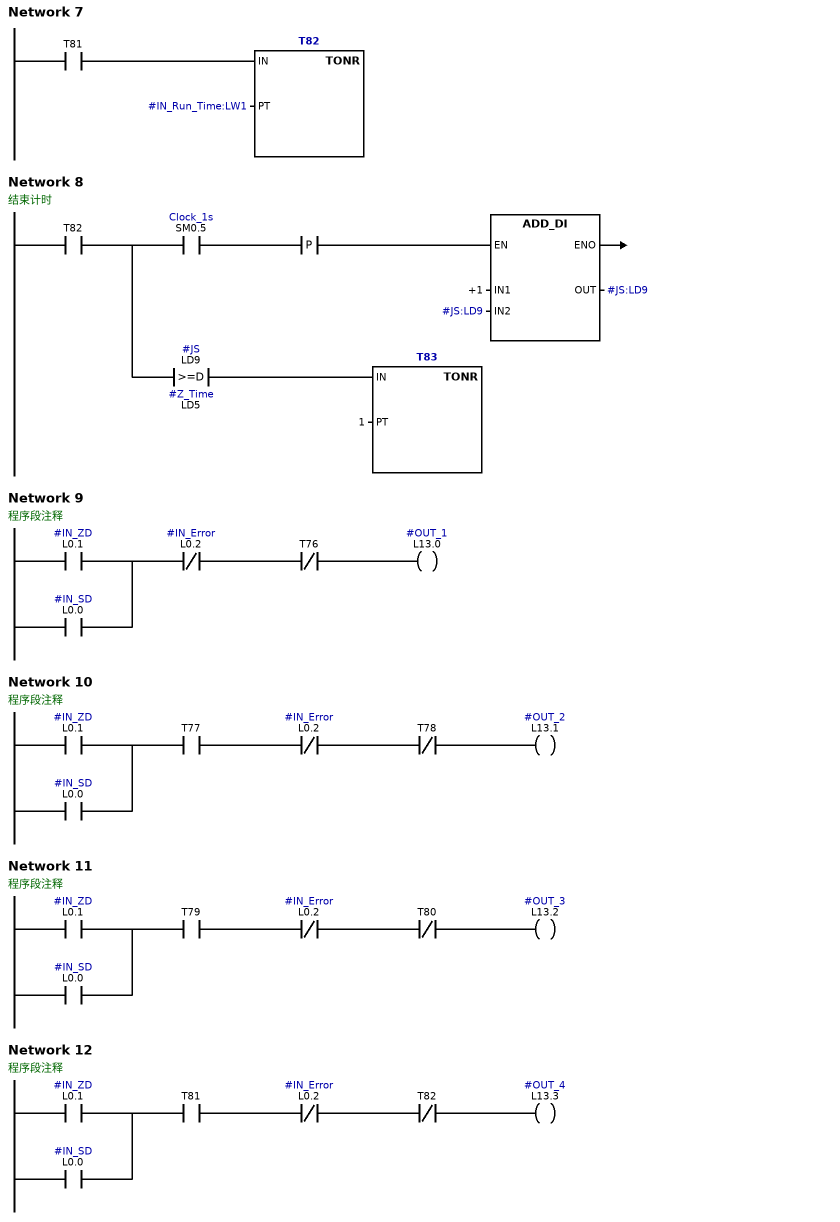
Network 7
LD     T81
TONR   T82, #IN_Run_Time:LW1
Network 8
// 结束计时
LD     T82
LPS
A      Clock_1s:SM0.5
EU
+D     +1, #JS:LD9
LPP
AD>=   #JS:LD9, #Z_Time:LD5
TONR   T83, 1
Network 9
//  程序段注释
LD     #IN_ZD:L0.1
O      #IN_SD:L0.0
AN     #IN_Error:L0.2
AN     T76
=      #OUT_1:L13.0
Network 10
//  程序段注释
LD     #IN_ZD:L0.1
O      #IN_SD:L0.0
A      T77
AN     #IN_Error:L0.2
AN     T78
=      #OUT_2:L13.1
Network 11
//  程序段注释
LD     #IN_ZD:L0.1
O      #IN_SD:L0.0
A      T79
AN     #IN_Error:L0.2
AN     T80
=      #OUT_3:L13.2
Network 12
//  程序段注释
LD     #IN_ZD:L0.1
O      #IN_SD:L0.0
A      T81
AN     #IN_Error:L0.2
AN     T82
=      #OUT_4:L13.3
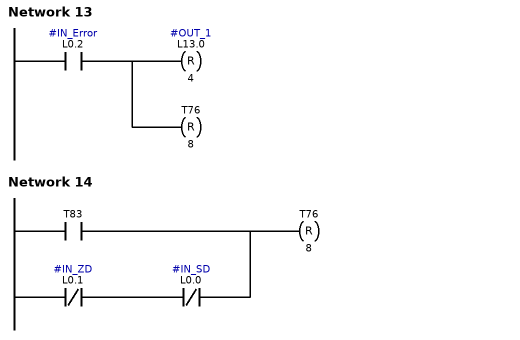
Network 13
LD     #IN_Error:L0.2
R      #OUT_1:L13.0, 4
R      T76, 8
Network 14
LD     T83
LDN    #IN_ZD:L0.1
AN     #IN_SD:L0.0
OLD
R      T76, 8
END_SUBROUTINE_BLOCK

SUBROUTINE_BLOCK 除铁器4组4:SBR88
TITLE=
VAR_INPUT
IN_SD:BOOL;	// L0.0 
IN_ZD:BOOL;	// L0.1 
IN_Error:BOOL;	// L0.2 
IN_Run_Time:INT;	// LW1 
IN_Stop_Time:INT;	// LW3 
Z_Time:DINT;	// LD5 
END_VAR
VAR_IN_OUT
JS:DINT;	// LD9 
END_VAR
VAR_OUTPUT
OUT_1:BOOL;	// L13.0 
OUT_2:BOOL;	// L13.1 
OUT_3:BOOL;	// L13.2 
OUT_4:BOOL;	// L13.3 
END_VAR
VAR
TP1:BOOL;	// L13.4 
TP2:BOOL;	// L13.5 
END_VAR
BEGIN
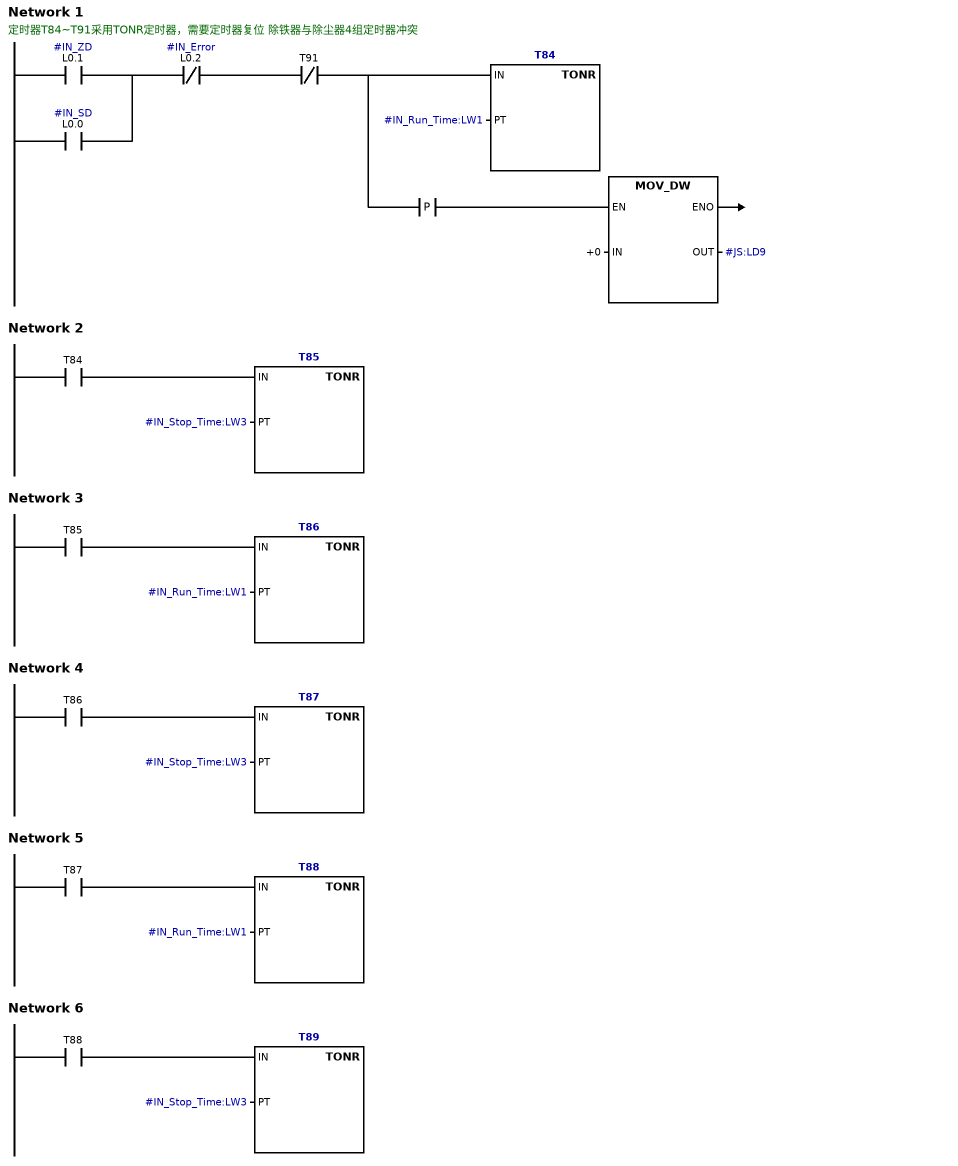
Network 1
// 定时器T84~T91采用TONR定时器，需要定时器复位 除铁器与除尘器4组定时器冲突
LD     #IN_ZD:L0.1
O      #IN_SD:L0.0
AN     #IN_Error:L0.2
AN     T91
TONR   T84, #IN_Run_Time:LW1
EU
MOVD   +0, #JS:LD9
Network 2
LD     T84
TONR   T85, #IN_Stop_Time:LW3
Network 3
LD     T85
TONR   T86, #IN_Run_Time:LW1
Network 4
LD     T86
TONR   T87, #IN_Stop_Time:LW3
Network 5
LD     T87
TONR   T88, #IN_Run_Time:LW1
Network 6
LD     T88
TONR   T89, #IN_Stop_Time:LW3
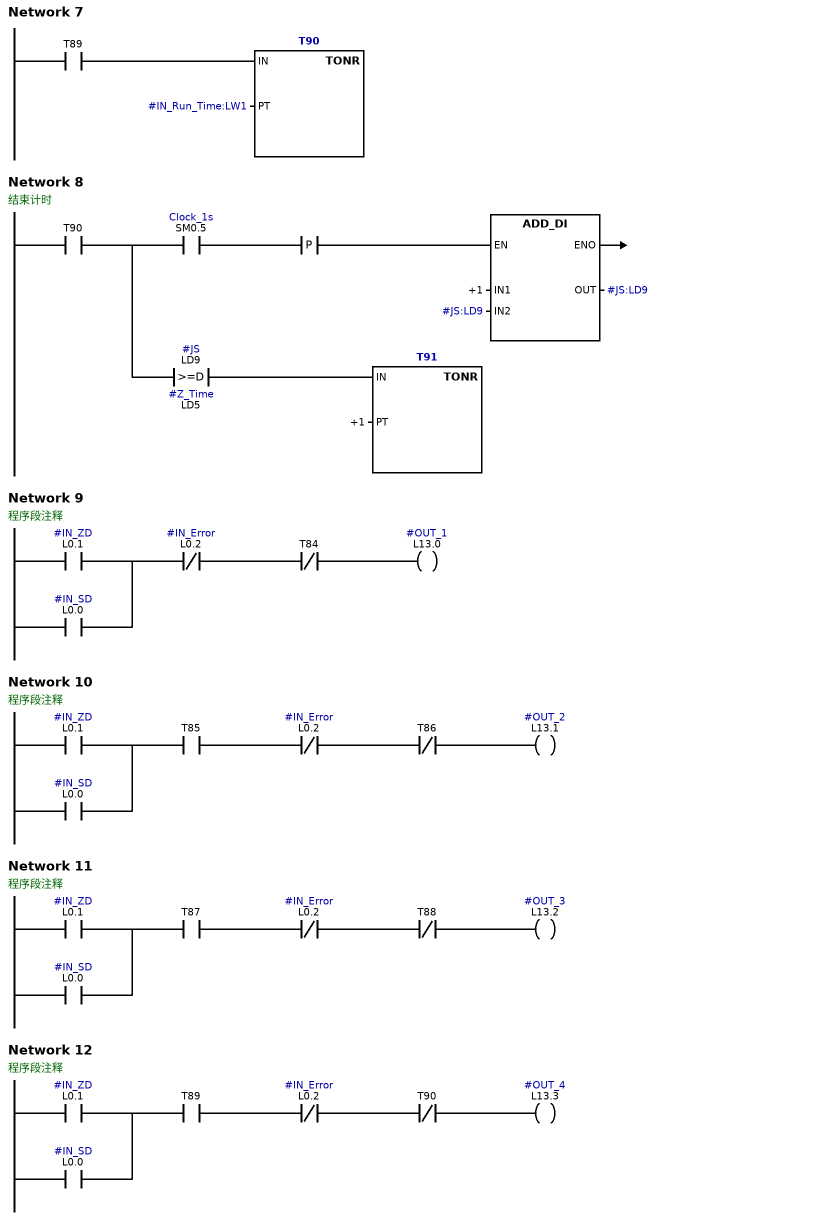
Network 7
LD     T89
TONR   T90, #IN_Run_Time:LW1
Network 8
// 结束计时
LD     T90
LPS
A      Clock_1s:SM0.5
EU
+D     +1, #JS:LD9
LPP
AD>=   #JS:LD9, #Z_Time:LD5
TONR   T91, +1
Network 9
//  程序段注释
LD     #IN_ZD:L0.1
O      #IN_SD:L0.0
AN     #IN_Error:L0.2
AN     T84
=      #OUT_1:L13.0
Network 10
//  程序段注释
LD     #IN_ZD:L0.1
O      #IN_SD:L0.0
A      T85
AN     #IN_Error:L0.2
AN     T86
=      #OUT_2:L13.1
Network 11
//  程序段注释
LD     #IN_ZD:L0.1
O      #IN_SD:L0.0
A      T87
AN     #IN_Error:L0.2
AN     T88
=      #OUT_3:L13.2
Network 12
//  程序段注释
LD     #IN_ZD:L0.1
O      #IN_SD:L0.0
A      T89
AN     #IN_Error:L0.2
AN     T90
=      #OUT_4:L13.3
